{attribute 'qualified_only'}
{attribute 'to_string'}
TYPE E_DGPD_SequenceStep :
(
    INIT,
    CHECK_OUT,
    MOVE_RET_TO_TARGET,
    MOVE_X_TO_TARGET,
    MOVE_Y_TO_TARGET,
    MOVE_Z_TO_TARGET,
    DONE,
    ERROR
);
END_TYPE

(* stored: Version 1.1.0.1
   DUT E_DGPD_SequenceStep: Id {d3314f97-48c6-4f62-9279-c41913c907ec} *)
